FUNCTION_BLOCK FB_MasterCamControl
VAR_INPUT
END_VAR
VAR_OUTPUT
END_VAR
VAR
//	fbMaster		: CAM_AXIS_BASE;
//	fbSlave_1		: CAM_AXIS_BASE;
//	fbSlave_2		: CAM_AXIS_BASE;
//	fbSlave_3		: CAM_AXIS_BASE;
//	fbSlave_4		: CAM_AXIS_BASE;
	mcHome			: MC_Home;
	bRunCams		: BOOL;
	
	bInitialized	: BOOL;
	bCamInDone		: BOOL;
END_VAR

//fbMaster.mRunCam(bRunCams);
//fbSlave_1.mRunCam(bRunCams);
//fbSlave_2.mRunCam(bRunCams);
//fbSlave_3.mRunCam(bRunCams);
//fbSlave_4.mRunCam(bRunCams);

// Reset Virtual Master Cam to 0 after 1 complete revolution
IF GVL.Master.NcToPlc.ModuloSetTurns = 1 AND NOT mcHome.Done THEN
	mcHome(
		Axis		:= GVL.Master,
		Execute		:= TRUE,
		Position	:= 0,
		HomingMode	:= MC_Direct);
ELSIF mcHome.Done THEN
	mcHome(Axis := GVL.Master, Execute := FALSE);
END_IF

METHOD mCamOut : BOOL
VAR_INPUT
	Execute		: BOOL;
END_VAR

VAR_INST
	CamOut		: MC_CamOut;
	
	nState		: INT;
	rtStart		: R_TRIG;
END_VAR
CASE nState OF
	0:
		rtStart(CLK := Execute);
		IF rtStart.Q THEN
			mCamOut		:= FALSE;
			nState		:= 5;
		END_IF
	5:
		CamOut(Slave := GVL.Slave_1, Execute := TRUE);
		IF CamOut.Done THEN
			CamOut(Slave := GVL.Slave_1, Execute := FALSE);
			nState		:= 15;
		END_IF
	15:
		CamOut(Slave := GVL.Slave_2, Execute := TRUE);
		IF CamOut.Done THEN
			CamOut(Slave := GVL.Slave_2, Execute := FALSE);
			nState		:= 20;
		END_IF
	20:
		CamOut(Slave := GVL.Slave_3, Execute := TRUE);
		IF CamOut.Done THEN
			CamOut(Slave := GVL.Slave_3, Execute := FALSE);
			nState		:= 25;
		END_IF
	25:
		CamOut(Slave := GVL.Slave_4, Execute := TRUE);
		IF CamOut.Done THEN
			CamOut(Slave := GVL.Slave_4, Execute := FALSE);
			nState		:= 30;
		END_IF
	30:
		mCamOut			:= TRUE;
		nState			:= 0;
END_CASE
END_METHOD

METHOD mHalt : BOOL
VAR_IN_OUT
	Execute		: BOOL;
END_VAR
VAR_INST
	HaltMaster	: MC_Halt;
	HaltSlave_1	: MC_Halt;
	HaltSlave_2	: MC_Halt;
	HaltSlave_3	: MC_Halt;
	HaltSlave_4	: MC_Halt;
END_VAR
HaltMaster(Axis := GVL.Master, Execute := Execute);
HaltSlave_1(Axis := GVL.Slave_1, Execute := Execute);
HaltSlave_2(Axis := GVL.Slave_2, Execute := Execute);
HaltSlave_3(Axis := GVL.Slave_3, Execute := Execute);
HaltSlave_4(Axis := GVL.Slave_4, Execute := Execute);

IF HaltMaster.Done AND HaltSlave_1.Done AND HaltSlave_2.Done AND HaltSlave_3.Done AND HaltSlave_4.Done THEN
	Execute := FALSE;
END_IF
END_METHOD

(* Move all axes to 0 position *)
METHOD mHomeAxes : BOOL
VAR_INPUT
	Execute			: BOOL;
END_VAR

VAR_INST
	MoveHome		: MC_MoveAbsolute;
	mcHome			: MC_Home;
	
	nState			: INT;
	rtStart			: R_TRIG;
END_VAR
CASE nState OF
	0:
		rtStart(CLK := Execute);
		IF rtStart.Q THEN
			mHomeAxes	:= FALSE;
			nState		:= 5;
		END_IF
	5:
		MoveHome(
			Axis		:= GVL.Slave_1,
			Execute		:= TRUE,
			Position	:= 0,
			Velocity	:= 2000);
		IF MoveHome.Done THEN
			MoveHome(Axis := GVL.Slave_1, Execute := FALSE);
			nState		:= 10;
		END_IF
	10:
		MoveHome(
			Axis		:= GVL.Slave_2,
			Execute		:= TRUE,
			Position	:= 0,
			Velocity	:= 2000);
		IF MoveHome.Done THEN
			MoveHome(Axis := GVL.Slave_2, Execute := FALSE);
			nState		:= 15;
		END_IF
	15:
		MoveHome(
			Axis		:= GVL.Slave_3,
			Execute		:= TRUE,
			Position	:= 0,
			Velocity	:= 2000);
		IF MoveHome.Done THEN
			MoveHome(Axis := GVL.Slave_3, Execute := FALSE);
			nState		:= 20;
		END_IF
	20:
		MoveHome(
			Axis		:= GVL.Slave_4,
			Execute		:= TRUE,
			Position	:= 0,
			Velocity	:= 2000);
		IF MoveHome.Done THEN
			MoveHome(Axis := GVL.Slave_4, Execute := FALSE);
			nState		:= 25;
		END_IF
	25:
		mcHome(
			Axis		:= GVL.Master,
			Execute		:= TRUE,
			Position	:= 0,
			HomingMode	:= MC_Direct);
		IF mcHome.Done THEN
			mcHome(Axis := GVL.Master, Execute := FALSE);
			nState		:= 30;
		END_IF
	30:
		mHomeAxes		:= TRUE;
		nState			:= 0;
END_CASE
END_METHOD

METHOD mInitialize : BOOL
VAR_INPUT
	Execute			: BOOL;
END_VAR
VAR_INST
	nState			: INT;
	rtStart			: R_TRIG;
END_VAR
CASE nState OF
	0:
		rtStart(CLK := Execute);
		IF rtStart.Q THEN
			bInitialized	:= FALSE;
			nState			:= 1;
		END_IF
	1:
		IF mCamOut(TRUE) THEN
			mCamOut(FALSE);
			nState			:= 5;
		END_IF
	5:
		IF mReset(TRUE) THEN
			mReset(FALSE);
			nState			:= 10;
		END_IF
	10:
		IF mPower(TRUE) THEN
			mPower(FALSE);
			nState			:= 15;
		END_IF
	15:
		IF mHomeAxes(TRUE) THEN
			mHomeAxes(FALSE);
			nState			:= 100;
		END_IF
	100:
		bInitialized		:= TRUE;
		nState				:= 0;
END_CASE
END_METHOD

METHOD mMultiCamIn : BOOL
VAR_INPUT
	Execute		: BOOL;
END_VAR

VAR_INST
	nState		: INT;
	rtStart		: R_TRIG;
	
	CamIn		: MC_CamIn;
	
	Options		: ST_CamInOptions;
END_VAR
CASE nState OF
	0:
		rtStart(CLK := Execute);
		IF rtStart.Q THEN
			Options.ActivationMode:= MC_CAMACTIVATION_INSTANTANEOUS;
			Options.InterpolationType:= MC_INTERPOLATIONTYPE_LINEAR;
			bCamInDone	:= FALSE;
			nState		:= 5;
		END_IF
	5:
		CamIn(
			Master		:= GVL.Master,
			Slave		:= GVL.Slave_1,
			Execute		:= TRUE,
 			StartMode	:= MC_STARTMODE_ABSOLUTE,
			Options		:= Options,
			CamTableID	:= 1);
		IF CamIn.InSync THEN
			CamIN(Master:= GVL.Master, Slave:= GVL.Slave_1, Execute:= FALSE);
			nState		:= 10;
		END_IF
	10:
		CamIn(
			Master		:= GVL.Master,
			Slave		:= GVL.Slave_2,
			Execute		:= TRUE,
			StartMode	:= MC_STARTMODE_ABSOLUTE,
			Options		:= Options,
			CamTableID	:= 2);
		IF CamIn.InSync THEN
			CamIN(Master:= GVL.Master, Slave:= GVL.Slave_2, Execute:= FALSE);
			nState		:= 15;
		END_IF
	15:
		CamIn(
			Master		:= GVL.Master,
			Slave		:= GVL.Slave_3,
			Execute		:= TRUE,
			StartMode	:= MC_STARTMODE_ABSOLUTE,
			Options		:= Options,
			CamTableID	:= 3);
		IF CamIn.InSync THEN
			CamIN(Master:= GVL.Master, Slave:= GVL.Slave_3, Execute:= FALSE);
			nState		:= 20;
		END_IF
	20:
		CamIn(
			Master		:= GVL.Master,
			Slave		:= GVL.Slave_4,
			Execute		:= TRUE,
			StartMode	:= MC_STARTMODE_ABSOLUTE,
			Options		:= Options,
			CamTableID	:= 4);
		IF CamIn.InSync THEN
			CamIN(Master:= GVL.Master, Slave:= GVL.Slave_4, Execute:= FALSE);
			nState		:= 25;
		END_IF
	25:
		bCamInDone		:= TRUE;
		nState			:= 0;
END_CASE
END_METHOD

METHOD mPower : BOOL
VAR_INPUT
	Execute			: BOOL;
END_VAR
VAR_INST
	nState			: INT;
	rtStart			: R_TRIG;
	
	PowerMaster				: MC_Power;
	PowerSlave_1			: MC_Power;
	PowerSlave_2			: MC_Power;
	PowerSlave_3			: MC_Power;
	PowerSlave_4			: MC_Power;
END_VAR
CASE nState OF
	0:
		rtStart(CLK := Execute);
		IF rtStart.Q THEN
			mPower			:= FALSE;
			nState			:= 5;
		END_IF
	5:
		PowerMaster(
			Axis			:= GVL.Master,
			Enable			:= TRUE,
			Enable_Positive	:= TRUE,
			Enable_Negative	:= TRUE);
		IF PowerMaster.Status THEN			// Status = Done (BOOL)
			nState			:= 10;
		END_IF
	10:
		PowerSlave_1(
			Axis			:= GVL.Slave_1,
			Enable			:= TRUE,
			Enable_Positive	:= TRUE,
			Enable_Negative	:= TRUE);
		IF PowerSlave_1.Status THEN
			nState			:= 15;
		END_IF
	15:
		PowerSlave_2(
			Axis			:= GVL.Slave_2,
			Enable			:= TRUE,
			Enable_Positive	:= TRUE,
			Enable_Negative	:= TRUE);
		IF PowerSlave_2.Status THEN
			nState			:= 20;
		END_IF
	20:
		PowerSlave_3(
			Axis			:= GVL.Slave_3,
			Enable			:= TRUE,
			Enable_Positive	:= TRUE,
			Enable_Negative	:= TRUE);
		IF PowerSlave_3.Status THEN
			nState			:= 25;
		END_IF
	25:
		PowerSlave_4(
			Axis			:= GVL.Slave_4,
			Enable			:= TRUE,
			Enable_Positive	:= TRUE,
			Enable_Negative	:= TRUE);
		IF PowerSlave_4.Status THEN
			nState			:= 100;
		END_IF
	100:
		mPower				:= TRUE;
		nState				:= 0;
END_CASE
END_METHOD

METHOD mReset : BOOL
VAR_INPUT
	Execute		: BOOL;
END_VAR
VAR_INST
//	ResetMaster	: MC_Reset;
//	ResetSlave_1: MC_Reset;
//	ResetSlave_2: MC_Reset;
//	ResetSlave_3: MC_Reset;
//	ResetSlave_4: MC_Reset;
	Reset		: MC_Reset;	

	nState		: INT;
	rtStart		: R_TRIG;
END_VAR
CASE nState OF
	0:
		rtStart(CLK := Execute);
		IF rtStart.Q THEN
			mReset	:= FALSE;
			nState	:= 10;
		END_IF
	10:
		Reset(Axis := GVL.Master, Execute := Execute);
		IF Reset.Done THEN
			Reset(Axis := GVL.Master, Execute := FALSE);
			nState	:= 15;
		END_IF
	15:
		Reset(Axis := GVL.Slave_1, Execute := Execute);
		IF Reset.Done THEN
			Reset(Axis := GVL.Slave_1, Execute := FALSE);
			nState	:= 20;
		END_IF
	20:
		Reset(Axis := GVL.Slave_2, Execute := Execute);
		IF Reset.Done THEN
			Reset(Axis := GVL.Slave_2, Execute := FALSE);
			nState	:= 25;
		END_IF
	25:
		Reset(Axis := GVL.Slave_3, Execute := Execute);
		IF Reset.Done THEN
			Reset(Axis := GVL.Slave_3, Execute := FALSE);
			nState	:= 30;
		END_IF
	30:
		Reset(Axis := GVL.Slave_4, Execute := Execute);
		IF Reset.Done THEN
			Reset(Axis := GVL.Slave_4, Execute := FALSE);
			nState	:= 35;
		END_IF
	35:
		mReset		:= TRUE;
		nState		:= 0;
END_CASE


//ResetMaster(Axis := Master, Execute := Execute);
//ResetSlave_1(Axis := Slave_1, Execute := Execute);
//ResetSlave_2(Axis := Slave_2, Execute := Execute);
//ResetSlave_3(Axis := Slave_3, Execute := Execute);
//ResetSlave_4(Axis := Slave_4, Execute := Execute);

//IF ResetMaster.Done AND ResetSlave_1.Done AND ResetSlave_2.Done AND ResetSlave_3.Done AND ResetSlave_4.Done THEN
//	Execute	:= FALSE;
//END_IF
END_METHOD

METHOD mRun : BOOL
VAR_INPUT
END_VAR
VAR_IN_OUT
	bMasterRun		: BOOL;
END_VAR
VAR_INST
	nState			: INT;
	rtRerun			: R_TRIG;
	
	MoveMaster 		: MC_MoveVelocity;
	
	MoveSlave_1		: MC_MoveAbsolute;
	MoveSlave_2		: MC_MoveAbsolute;
	MoveSlave_3		: MC_MoveAbsolute;
	MoveSlave_4		: MC_MoveAbsolute;
END_VAR
IF bMasterRun THEN
	MoveMaster(
		Axis		:= GVL.Master,
		Execute		:= TRUE,
		Velocity	:= GVL.rMasterVel,
		Direction	:= MC_Positive_Direction);
	IF MoveMaster.InVelocity THEN
		MoveMaster(Axis := GVL.Master, Execute := FALSE);
		bMasterRun	:= FALSE;
	END_IF
END_IF

MoveSlave_1(
	Axis		:= GVL.Slave_1,
	Execute		:= bRunCams,
	Position	:= 0,
	Velocity	:= 1000);
MoveSlave_2(
	Axis		:= GVL.Slave_2,
	Execute		:= bRunCams,
	Position	:= 0,
	Velocity	:= 1000);
MoveSlave_3(
	Axis		:= GVL.Slave_3,
	Execute		:= bRunCams,
	Position	:= 0,
	Velocity	:= 1000);
MoveSlave_4(
	Axis		:= GVL.Slave_4,
	Execute		:= bRunCams,
	Position	:= 0,
	Velocity	:= 1000);
END_METHOD

PROPERTY pCamInDone : BOOL
GET
pCamInDone := bCamInDone;
END_GET
END_PROPERTY

PROPERTY pInitialized : BOOL
GET
pInitialized := bInitialized;
END_GET
END_PROPERTY

PROPERTY pRunCams : BOOL
GET
pRunCams := bRunCams;
END_GET
SET
bRunCams := pRunCams;
END_SET
END_PROPERTY

END_FUNCTION_BLOCK

(* stored: Version 1.1.0.1, ProductVersion 3.1.4024.15
   POU FB_MasterCamControl: Id {563d04a1-1878-491b-b5bf-d0acddfa2dc7}, SpecialFunc None
   Method mCamOut: Id {fec35e8c-ce4a-4b90-be2e-5dd8bb43044e}
   Method mHalt: Id {a03e96ed-f4ca-4d55-a866-0c612669a200}
   Method mHomeAxes: Id {3dafe4fd-36db-4d2b-a1a0-e571e50f84c5}
   Method mInitialize: Id {9573a738-c4c6-41ee-bdc4-c7aa6dc47070}
   Method mMultiCamIn: Id {ae1371a6-3971-4de4-9f5e-3ff07e00bbd9}
   Method mPower: Id {df25cbad-15f3-45a6-8254-8d21a94a4d9a}
   Method mReset: Id {4f7ff489-d1c4-45ad-91f1-fdfcac150328}
   Method mRun: Id {f142f0e0-c512-4da0-9a9a-fab148c051f5}
   Property pCamInDone: Id {725efcde-17db-48a1-9037-d6cb9b573392}
   Get Get: Id {648050a1-777f-4a77-bc0e-4ca49d004044}
   Property pInitialized: Id {b7815016-286e-4928-ae20-4eea446711b1}
   Get Get: Id {6238a259-6a2d-4043-bf00-fd4abc03693d}
   Property pRunCams: Id {3eb23a41-149a-4da0-b761-d62043bf919b}
   Get Get: Id {2130c9d1-da89-4479-9d0d-be8f500b0a03}
   Set Set: Id {ce7f989a-80be-4e25-8f47-44b00e4ea335} *)
